{attribute 'linkalways'} 
{attribute 'no_explicit_call' := 'This FB is a CLASS and must be accessed using methods or properties'}
{attribute 'enable_dynamic_creation'}
FUNCTION_BLOCK INTERNAL MoveAbsoluteCommand EXTENDS MoveCommand
VAR
	_fb : MC_MoveAbsolute;
	_position : LREAL;
END_VAR

METHOD FB_init : BOOL
VAR_INPUT
	bInitRetains : BOOL; // if TRUE, the retain variables are initialized (warm start / cold start)
	bInCopyCode : BOOL;  // if TRUE, the instance afterwards gets moved into the copy code (online change)
	axis : I_Axis;
	position : LREAL;
	velocity : LREAL;
	acceleration : LREAL;
	deceleration : LREAL;
	jerk : LREAL;
	bufferMode : AxisBufferMode;
END_VAR
_axis := axis;
_position := position;
_velocity := velocity;
_acceleration := acceleration;
_deceleration := deceleration;
_jerk := jerk;
_bufferMode := bufferMode;
END_METHOD

METHOD PROTECTED WhileBusy
VAR_INPUT
	CommandState : I_CommandBusyState;
END_VAR
_fb(
	Axis := _axis._InternalAxisRef,
	Execute := TRUE,
	Position := _position,
	Velocity := _velocity,
	Acceleration := _acceleration,
	Deceleration := _deceleration,
	Jerk := _jerk,
	BufferMode := _bufferMode
);

IF _fb.Busy THEN
	RETURN;
END_IF

IF _fb.CommandAborted THEN
	_fb(Axis := _axis._InternalAxisRef, Execute := FALSE);
	CommandState.SetAborting();
	RETURN;
END_IF

IF _fb.Error THEN
	_fb(Axis := _axis._InternalAxisRef, Execute := FALSE);
	CommandState.SetError(_fb.ErrorID);
	RETURN;
END_IF

_fb(Axis := _axis._InternalAxisRef, Execute := FALSE);
CommandState.SetDone();
END_METHOD

END_FUNCTION_BLOCK

(* stored: Version 1.1.0.1, ProductVersion 3.1.4024.12
   POU MoveAbsoluteCommand: Id {f2bf5d21-cab0-4b95-ae14-e4f31a338d45}, SpecialFunc None
   Folder Constructor: Id {ac24e1f2-7bc9-4ec0-98ca-84b69e8381bb}
   Method FB_init: Id {304daf3f-1f91-4d37-b06b-2471eab077be}
   Method WhileBusy: Id {51d7502a-7fb5-4811-b305-b98249d64ac5} *)
